{attribute 'qualified_only'}
VAR_GLOBAL
    stTerm1_EK1100     : ST_EK1100;
    stTerm2_EL6070     : ST_EL6070;
    stTerm3_EL6910     : ST_EL6910;
    stTerm4_EL1918     : ST_EL1918;
    stTerm5_EL1918     : ST_EL1918;
    stTerm6_EL2904     : ST_EL2904;
    stTerm7_EL1809     : ST_EL1809;
    stTerm8_EL1809     : ST_EL1809;
    stTerm9_EL2809     : ST_EL2809;
    stTerm10_EL2809    : ST_EL2809;
    stTerm11_EL3058    : ST_EL3058;
    stTerm12_EL3064    : ST_EL3064;
    stTerm13_EL9410    : ST_EL9410;
	stTerm14_EL3064	   : ST_EL3064;
    stTerm15_EL6652    : ST_EL6652;
	stTerm33_EL3314    : ST_EL3314;
END_VAR

(* stored: Version 1.1.0.1, ProductVersion 3.1.4026.18
   GVL GVL_EtherCAT: Id {0c762596-e7cb-44aa-8f7d-0709ef4bd060} *)
